// TIA Portal V19 export
DATA_BLOCK "LPNDR_Readportinfo"   // DB33
// stored: InstanceOfName LPNDR_ReadGlobalInfo_2, InstanceOfType FB
"LPNDR_ReadGlobalInfo_2"
   // VAR_INPUT
   //    execute : Bool;
   //    hwId : HW_IO;
   //    mode : Int;
   // END_VAR
   // VAR_OUTPUT
   //    busy : Bool;
   //    done : Bool;
   //    error : Bool;
   //    status : Word;
   // END_VAR
   // VAR_IN_OUT
   //    DataRecord : Variant;
   // END_VAR
   // VAR
   //    InstReadRecord { S7_SetPoint := 'True'} : RDREC;
   //    statReadRecord { ExternalAccessible := 'False'; ExternalVisible := 'False'; ExternalWritable := 'False'} : Array[0..4175] of Byte;
   //    statReadRecordLength : UInt;
   //    statReadRecordRequest : Bool;
   //    statOldExecute : Bool;
   //    statPDInterfaceMrpDataReal : UInt;
   //    statPDPortMrpDataReal : UInt;
   //    statPDInterfaceDataReal : UInt;
   //    statPDPortDataReal : UInt;
   //    statPDPortStatistic : UInt;
   //    statUnknown : UInt;
   //    statInterfaceInformation { S7_SetPoint := 'True'} : "LPNDR_typeInterfaceInformation";
   //    statPortInformation { S7_SetPoint := 'True'} : Array[1..52] of "LPNDR_typePortInformation";
   //    statPortLinkState { S7_SetPoint := 'True'} : Array[1..52] of "LPNDR_typePortLinkState";
   //    statPortStatistic { S7_SetPoint := 'True'} : Array[1..52] of "LPNDR_typePortStatistic";
   //    statBusy { S7_SetPoint := 'True'} : Bool;
   // END_VAR
BEGIN
END_DATA_BLOCK
